PROGRAM P5_01_EnableControls
VAR
	tonDisableNext			:TON;
	tonDisablePrev			:TON;
	tonDelayLid				:TON;
END_VAR
VAR // added by the converter: edge detectors and wires of the graphical bodies
    _w1 : BOOL;
END_VAR

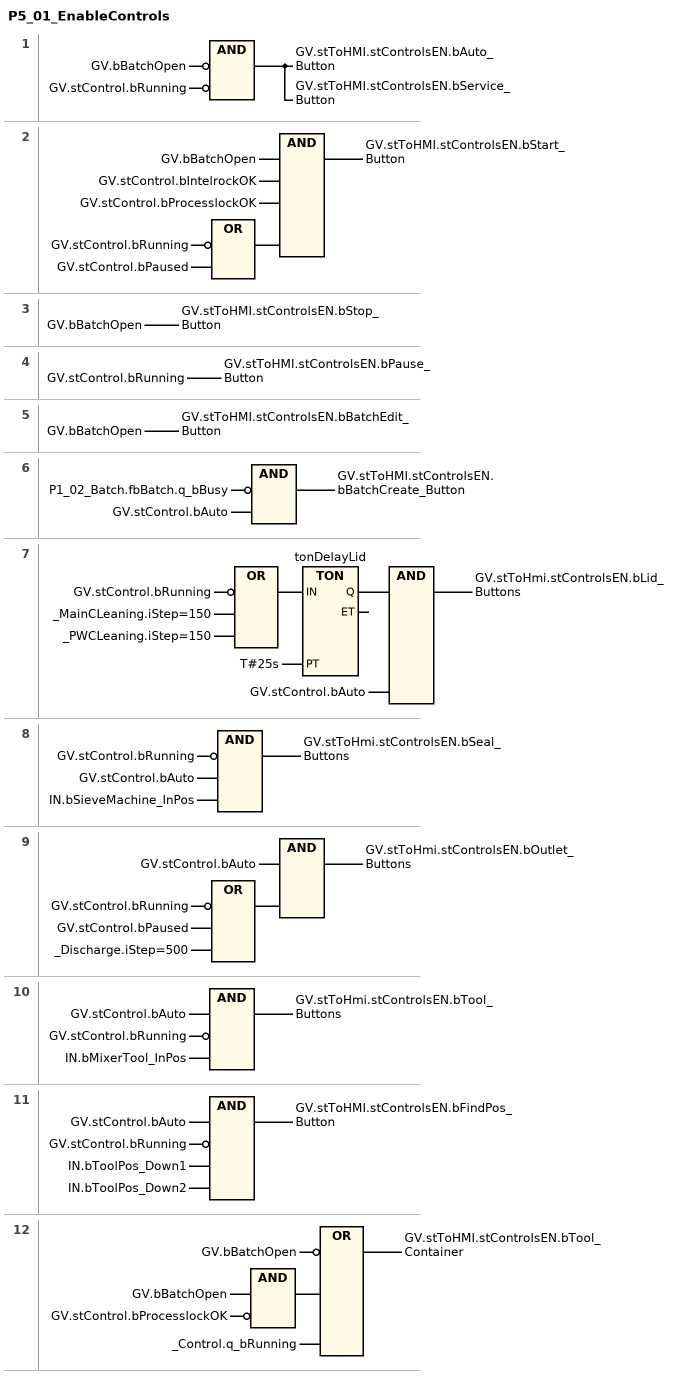
// NETWORK 1
_w1 := NOT GV.bBatchOpen AND NOT GV.stControl.bRunning;
GV.stToHMI.stControlsEN.bAuto_Button := _w1;
GV.stToHMI.stControlsEN.bService_Button := _w1;

// NETWORK 2
GV.stToHMI.stControlsEN.bStart_Button := GV.bBatchOpen AND GV.stControl.bIntelrockOK AND GV.stControl.bProcesslockOK AND (NOT GV.stControl.bRunning OR GV.stControl.bPaused);

// NETWORK 3
GV.stToHMI.stControlsEN.bStop_Button := GV.bBatchOpen;

// NETWORK 4
GV.stToHMI.stControlsEN.bPause_Button := GV.stControl.bRunning;

// NETWORK 5
GV.stToHMI.stControlsEN.bBatchEdit_Button := GV.bBatchOpen;

// NETWORK 6
GV.stToHMI.stControlsEN.bBatchCreate_Button := NOT P1_02_Batch.fbBatch.q_bBusy AND GV.stControl.bAuto;

// NETWORK 7
tonDelayLid(IN := NOT GV.stControl.bRunning OR (_MainCLeaning.iStep=150) OR (_PWCLeaning.iStep=150), PT := T#25s); // TON
GV.stToHmi.stControlsEN.bLid_Buttons := tonDelayLid.Q AND GV.stControl.bAuto;

// NETWORK 8
GV.stToHmi.stControlsEN.bSeal_Buttons := NOT GV.stControl.bRunning AND GV.stControl.bAuto AND IN.bSieveMachine_InPos;

// NETWORK 9
GV.stToHmi.stControlsEN.bOutlet_Buttons := GV.stControl.bAuto AND (NOT GV.stControl.bRunning OR GV.stControl.bPaused OR (_Discharge.iStep=500));

// NETWORK 10
GV.stToHmi.stControlsEN.bTool_Buttons := GV.stControl.bAuto AND NOT GV.stControl.bRunning AND IN.bMixerTool_InPos;

// NETWORK 11
GV.stToHMI.stControlsEN.bFindPos_Button := GV.stControl.bAuto AND NOT GV.stControl.bRunning AND IN.bToolPos_Down1 AND IN.bToolPos_Down2;

// NETWORK 12
GV.stToHMI.stControlsEN.bTool_Container := NOT GV.bBatchOpen OR GV.bBatchOpen AND NOT GV.stControl.bProcesslockOK OR _Control.q_bRunning;

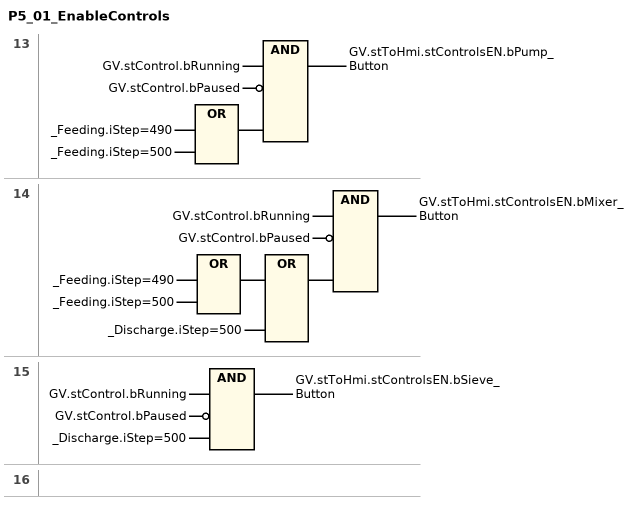
// NETWORK 13
GV.stToHmi.stControlsEN.bPump_Button := GV.stControl.bRunning AND NOT GV.stControl.bPaused AND ((_Feeding.iStep=490) OR (_Feeding.iStep=500));

// NETWORK 14
GV.stToHmi.stControlsEN.bMixer_Button := GV.stControl.bRunning AND NOT GV.stControl.bPaused AND (((_Feeding.iStep=490) OR (_Feeding.iStep=500)) OR (_Discharge.iStep=500));

// NETWORK 15
GV.stToHmi.stControlsEN.bSieve_Button := GV.stControl.bRunning AND NOT GV.stControl.bPaused AND (_Discharge.iStep=500);

// NETWORK 16

END_PROGRAM

(* stored: Version 1.1.0.1, ProductVersion 3.1.4026.13
   POU P5_01_EnableControls: Id {03708f81-cf31-4f21-abf9-33628c5a6011}, SpecialFunc None *)
